{attribute 'qualified_only' := ''}
{attribute 'strict' := ''}
TYPE eFirmerOperatingState :
(
	eNoInfo := 0,
	eOff := 1,
	eSleeping := 2,
	eStarting := 3,
	eMppt := 4,
	eThrottled := 5,
	eShuttingDown := 6,
	eFault := 7,
	eStandby := 8
);
END_TYPE

(* stored: Version 1.1.0.1, ProductVersion 3.1.4024.11
   DUT eFirmerOperatingState: Id {ce499511-6439-43f2-b2cc-8ed79f3ea140} *)
